TYPE "PPrf_SetUp"
VERSION : 0.1
// Block: PPrf_SetUp
   STRUCT
      Aut : PPrf_SetUp_Aut;
      Man : PPrf_SetUp_Man;
   END_STRUCT;

END_TYPE
